Staubli VAL3: getTrajItem.pgx

public program getTrajItem(TrajectoryItem& x_tTraj[] (dimensions=1), num x_nIndex (dimensions=1))
begin
  //
  // get all the FIELD
  //
  x_tTraj=pEditPoint.tData[x_nIndex].tSuper
end
